// Engineering-unit tag carried by analog IO config structs. Lets the HMI
// render the unit alongside the value without hard-coding the string at the
// caller. Extend by appending new enumerators at the end; existing codes
// are stable so historian / OPC tags do not shift.
//
// Last used enumerator: 32
{attribute 'qualified_only'}
{attribute 'strict'}
{attribute 'to_string'}
TYPE E_Unit :
(
    // Temperature
    DEGREE_CELSIUS                := 0,     // C
    DEGREE_FAHRENHEIT             := 31,    // F

    // Percentage & Level
    PERCENT                       := 1,

    // pH & Chemistry
    PH                            := 2,
    ORP                           := 3,     // mV - Oxidation Reduction Potential
    SOLIDS                        := 4,     // wt% - weight percent
    TURBIDITY                     := 5,     // NTU - Nephelometric Turbidity Units

    // Flow - Liquid (volumetric)
    CUBIC_METER_PER_HOUR          := 6,     // m3/hr
    LITER_PER_MINUTE              := 7,     // L/min
    STANDARD_LITER_PER_MINUTE     := 26,    // sL/min
    MILLILITER_PER_MINUTE         := 8,     // mL/min

    // Flow - Gas (volumetric)
    NORMAL_CUBIC_METER_PER_HOUR   := 9,     // Nm3/hr
    ACTUAL_LITERS_PER_MINUTE      := 30,    // ALPM

    // Gas monitoring
    PERCENT_LOWER_EXPLOSIVE_LIMIT := 27,    // %LEL

    // Mass flow / mass
    KILOGRAM_PER_HOUR             := 10,    // kg/hr
    KILOGRAM                      := 11,    // kg

    // Pressure
    KILOPASCAL                    := 12,    // kPa
    INCH_WATER_COLUMN             := 13,    // inWC
    PSIG                          := 14,    // psig - gauge pressure
    PSIA                          := 25,    // psia - absolute pressure

    // Density
    KILOGRAM_PER_CUBIC_METER      := 15,    // kg/m3

    // Electrical
    AMPS                          := 16,    // A
    VOLTS                         := 17,    // V
    MILLIVOLTS                    := 18,    // mV
    MICROVOLTS                    := 28,    // uV

    // Conductivity
    MICROSIEMENS_PER_CENTIMETER   := 19,    // uS/cm
    MILLISIEMENS_PER_CENTIMETER   := 20,    // mS/cm

    // Frequency & speed
    HERTZ                         := 21,    // Hz
    RPM                           := 22,    // RPM

    // Energy & power
    KILOWATT                      := 23,    // kW
    WATT                          := 32,    // W

    // Distance
    MILLIMETER                    := 24,    // mm

    // Quantity
    PPM                           := 29     // ppm
);
END_TYPE

(* stored: Version 1.1.0.1, ProductVersion 3.1.4026.12
   DUT E_Unit: Id {c0000030-0000-0000-0000-000000000002} *)
